(* PLC project Generated.project, CODESYS CODESYS V3.5 SP19 Patch 1 *)
(* stored: creationDateTime 2026-09-06T13:00:42.491081, modificationDateTime 2026-09-06T13:00:42.491081 *)

(* ═══════════════════════════════════════════════════════════════ 🎮 ST_WinchCmd — Commandes IHM pour un Treuil M1/M2 ─────────────────────────────────────────────────────────────── 🎨 Destiné au pilotage manuel et maintenance du treuil depuis l'IHM. ═══════════════════════════════════════════════════════════════ *)
TYPE ST_WinchCmd : STRUCT
  BtnAscent : BOOL;  (* ⬆️ Mouvement montee maintenu (mode boutons IHM, MAINT_N1 accessible) *)
  BtnDescent : BOOL;  (* ⬇️ Mouvement descente maintenu (mode boutons IHM, MAINT_N1 accessible) *)
  BtnReset : BOOL;  (* 🔑 Demande reset exposée par treuil ; agrégée dans le reset domaine partagé *)
  BtnHome : BOOL;  (* 🎯 Homing nominal si Couplé, unitaire si M1/M2 sélectionné en MAINT_N2 *)
  BtnConfirmCoherence : BOOL;  (* 🔓 Confirmation de cohérence au démarrage *)
  BtnInhibit : BOOL;  (* Bouton IHM inhibition treuil — mise en service, *)
  BtnHomingAtZero : BOOL;  (* Force le homing à 0 m (points codeur centre), *)
  BtnOverrideTopSoftware : BOOL;  (* Autorisation MAINTENUE de dépasser le FDC *)
  BtnLearnSpeed : BOOL;  (* 💾 Bit IHM lancer l'apprentissage passif des vitesses *)
END_STRUCT;
END_TYPE
